// TwinCAT 3 PLC project Ohjaus
// ProgramVersion: 3.1.4024.0
// libraries:
//   Tc2_Standard, * (Beckhoff Automation GmbH)
//   Tc2_System, * (Beckhoff Automation GmbH)
//   Tc3_Module, * (Beckhoff Automation GmbH)
//   VisuSymbols,3.5.10.0,System
// project tree:
//   / GlobalTextList.TcGTLO, PlcTask.TcTTO, Visualization Manager.TcVMO (not stored)
//   GVLs/ GVL.TcGVL, GVL_safety.TcGVL
//   POUs/ MAIN.TcPOU
//   POUs/Modules/ Handling.TcPOU, PickandPlace.TcPOU, Separating.TcPOU, Visu_handling.TcPOU, Sorting.TcPOU
//   VISUs/ Visualization.TcVIS
// real-time tasks:
//   TASK PlcTask: cycle T#10ms, priority 20, ADS port 350
// I/O:
//   DEVICE Device 1 (EtherCAT), AmsNetId 5.59.45.73.2.1
//     Term 1 (EK1200) [EK1200-5000 EtherCAT Power supply (2A E-Bus)]
//       Term 2 (EL1809) [EL1809 16Ch. Dig. Input 24V, 3ms]
//       Term 3 (EL2809) [EL2809 16Ch. Dig. Output 24V, 0.5A]
//       Term 4 (EL4021) [EL4021 1Ch. Ana. Output 4-20mA, 12bit]
//       Term 5 (EL3061) [EL3061 1Ch. Ana. Input 0-10V]
//       Term 6 (EL4021) [EL4021 1Ch. Ana. Output 4-20mA, 12bit]
//       Term 7 (EL2809) [EL2809 16Ch. Dig. Output 24V, 0.5A]
//       Term 8 (EL1809) [EL1809 16Ch. Dig. Input 24V, 3ms]
//       Term 9 (EL6900) [EL6900, TwinSAFE PLC]
//       Term 10 (EL1904) [EL1904, 4 Ch. Safety Input 24V, TwinSAFE]
//         modules: Module 1 (FSOES)
//       Term 11 (EL2904) [EL2904, 4 Ch. Safety Output 24V, 0.5A, TwinSAFE]
//         modules: Module 1 (FSOES), Module 2 (DO)
//       Term 12 (EL9011) [EL9011 End Terminal]
//   DEVICE Device 3 (NOV-DP-RAM)
// variable links:
//   Device 1 (EtherCAT) <-> Device 1 (EtherCAT)/Term 1 (EK1200)/Term 10 (EL1904)
//     Term 1 (EK1200)/Term 9 (EL6900)/ConnectionOutputs/Message_5 RxPDO <-> Module 1 (FSOES)/TxPDO/FSOE
//   Device 1 (EtherCAT) <-> Device 1 (EtherCAT)/Term 1 (EK1200)/Term 11 (EL2904)
//     Term 1 (EK1200)/Term 9 (EL6900)/ConnectionOutputs/Message_6 RxPDO <-> Module 1 (FSOES)/TxPDO/FSOE
//   Device 1 (EtherCAT) <-> Device 1 (EtherCAT)/Term 1 (EK1200)/Term 9 (EL6900)
//     Term 1 (EK1200)/Term 10 (EL1904)/Module 1 (FSOES)/RxPDO/FSOE <-> ConnectionInputs/Message_5 TxPDO
//     Term 1 (EK1200)/Term 11 (EL2904)/Module 1 (FSOES)/RxPDO/FSOE <-> ConnectionInputs/Message_6 TxPDO
//   Ohjaus/Ohjaus Instance <-> Device 1 (EtherCAT)/Term 1 (EK1200)/Term 2 (EL1809)
//     PlcTask Inputs/GVL.X1_I0 <-> Channel 9/Input
//     PlcTask Inputs/GVL.X1_I1 <-> Channel 10/Input
//     PlcTask Inputs/GVL.X1_I2 <-> Channel 13/Input
//     PlcTask Inputs/GVL.X1_I3 <-> Channel 14/Input
//     PlcTask Inputs/GVL.X1_I4 <-> Channel 15/Input
//     PlcTask Inputs/GVL.X1_I5 <-> Channel 16/Input
//     PlcTask Inputs/GVL.X1_I6 <-> Channel 1/Input
//     PlcTask Inputs/GVL.X1_I7 <-> Channel 2/Input
//     PlcTask Inputs/GVL.X2_I0 <-> Channel 3/Input
//     PlcTask Inputs/GVL.X2_I1 <-> Channel 4/Input
//     PlcTask Inputs/GVL.X2_I2 <-> Channel 5/Input
//     PlcTask Inputs/GVL.X2_I4 <-> Channel 6/Input
//     PlcTask Inputs/GVL.X2_I5 <-> Channel 7/Input
//     PlcTask Inputs/GVL_safety.Relay1_EDM <-> Channel 11/Input
//     PlcTask Inputs/GVL_safety.Start_button <-> Channel 12/Input
//   Ohjaus/Ohjaus Instance <-> Device 1 (EtherCAT)/Term 1 (EK1200)/Term 3 (EL2809)
//     PlcTask Outputs/GVL.X1_00 <-> Channel 5/Output
//     PlcTask Outputs/GVL.X1_01 <-> Channel 6/Output
//     PlcTask Outputs/GVL.X1_02 <-> Channel 7/Output
//     PlcTask Outputs/GVL.X1_03 <-> Channel 9/Output
//     PlcTask Outputs/GVL.X1_04 <-> Channel 10/Output
//     PlcTask Outputs/GVL.X1_05 <-> Channel 11/Output
//     PlcTask Outputs/GVL.X1_06 <-> Channel 12/Output
//     PlcTask Outputs/GVL.X1_07 <-> Channel 13/Output
//     PlcTask Outputs/GVL.X2_00 <-> Channel 14/Output
//     PlcTask Outputs/GVL.X2_01 <-> Channel 15/Output
//     PlcTask Outputs/GVL.X2_02 <-> Channel 16/Output
//     PlcTask Outputs/GVL.X4_00 <-> Channel 1/Output
//     PlcTask Outputs/GVL.X4_01 <-> Channel 2/Output
//     PlcTask Outputs/GVL.X4_02 <-> Channel 3/Output
//     PlcTask Outputs/GVL.X4_03 <-> Channel 4/Output
//     PlcTask Outputs/GVL.X4_07 <-> Channel 8/Output
//   Ohjaus/Ohjaus Instance <-> Device 1 (EtherCAT)/Term 1 (EK1200)/Term 7 (EL2809)
//     PlcTask Outputs/GVL.Safety_startpulse <-> Channel 6/Output
//     PlcTask Outputs/GVL.X2_03 <-> Channel 9/Output
//     PlcTask Outputs/GVL.X2_04 <-> Channel 10/Output
//     PlcTask Outputs/GVL.X2_05 <-> Channel 11/Output
//     PlcTask Outputs/GVL.X2_06 <-> Channel 12/Output
//     PlcTask Outputs/GVL.X2_07 <-> Channel 13/Output
//     PlcTask Outputs/GVL.X3_00 <-> Channel 1/Output
//     PlcTask Outputs/GVL.X3_01 <-> Channel 2/Output
//     PlcTask Outputs/GVL.X3_02 <-> Channel 3/Output
//     PlcTask Outputs/GVL.X3_03 <-> Channel 4/Output
//     PlcTask Outputs/GVL.X3_04 <-> Channel 5/Output
//     PlcTask Outputs/GVL.X3_06 <-> Channel 7/Output
//     PlcTask Outputs/GVL.X3_07 <-> Channel 8/Output
//   Ohjaus/Ohjaus Instance <-> Device 1 (EtherCAT)/Term 1 (EK1200)/Term 8 (EL1809)
//     PlcTask Inputs/GVL.X2_I6 <-> Channel 9/Input
//     PlcTask Inputs/GVL.X2_I7 <-> Channel 10/Input
//     PlcTask Inputs/GVL.X3_I0 <-> Channel 1/Input
//     PlcTask Inputs/GVL.X3_I1 <-> Channel 2/Input
//     PlcTask Inputs/GVL.X3_I2 <-> Channel 3/Input
//     PlcTask Inputs/GVL.X3_I4 <-> Channel 4/Input
//     PlcTask Inputs/GVL.X3_I5 <-> Channel 5/Input
//     PlcTask Inputs/GVL.X3_I6 <-> Channel 6/Input
//     PlcTask Inputs/GVL.X4_I0 <-> Channel 11/Input
//     PlcTask Inputs/GVL.X4_I1 <-> Channel 12/Input
//     PlcTask Inputs/GVL.X4_I2 <-> Channel 13/Input
//     PlcTask Inputs/GVL.X4_I3 <-> Channel 14/Input
//     PlcTask Inputs/GVL.X4_I4 <-> Channel 15/Input
//     PlcTask Inputs/GVL.X4_I5 <-> Channel 16/Input
//     PlcTask Inputs/GVL_safety.Safety_Restart <-> Channel 8/Input
//     PlcTask Inputs/MAIN.IbEStopReset <-> Channel 7/Input
//   Ohjaus/Ohjaus Instance <-> Device 1 (EtherCAT)/Term 1 (EK1200)/Term 9 (EL6900)
//     PlcTask Inputs/GVL_safety.Com_Err <-> StandardInputs/Standard Out Var 13
//     PlcTask Inputs/GVL_safety.FB_Err <-> StandardInputs/Standard Out Var 12
//     PlcTask Inputs/GVL_safety.Out_Err <-> StandardInputs/Standard Out Var 14
//     PlcTask Inputs/GVL_safety.Start_pulse <-> StandardInputs/Standard Out Var 9
//     PlcTask Inputs/MAIN.IbEStopError <-> StandardInputs/Standard Out Var 10
//     PlcTask Outputs/GVL_safety.Safety_RUNSTOP <-> StandardOutputs/Standard In Var 11
//     PlcTask Outputs/MAIN.QbEStopReset <-> StandardOutputs/Standard In Var 8
//     PlcTask Outputs/MAIN.QbSafetyErrAck <-> StandardOutputs/Standard In Var 2
//     PlcTask Outputs/MAIN.relay1 <-> StandardOutputs/Standard In Var 7

CONFIGURATION Ohjaus
    RESOURCE PLC ON TwinCAT3
        TASK PlcTask(INTERVAL := T#10ms, PRIORITY := 20);
        PROGRAM MAIN WITH PlcTask : MAIN;
        PROGRAM Visu_handling WITH PlcTask : Visu_handling;
        PROGRAM PickandPlace WITH PlcTask : PickandPlace;
        PROGRAM Sorting WITH PlcTask : Sorting;
        PROGRAM Handling WITH PlcTask : Handling;
        PROGRAM Separating WITH PlcTask : Separating;
    END_RESOURCE
END_CONFIGURATION

// ---- GVLs/GVL.TcGVL
{attribute 'qualified_only'}
VAR_GLOBAL
	X1_I0 AT %I* : BOOL; // Part available
	X1_I1 AT %I* : BOOL; // Mini-slide rectracted
	X1_I2 AT %I* : BOOL; // Mini-slide extended
	X1_I3 AT %I* : BOOL; // Mini-slide up
	X1_I4 AT %I* : BOOL; // Workpiece picked up
	X1_I5 AT %I* : BOOL; // Workpiece at processing position
	X1_I6 AT %I* : BOOL; // No workpiece at conveyor end
	X1_I7 AT %I* : BOOL; // Downstream station free
	X2_I0 AT %I* : BOOL; // Workpeace available
	X2_I1 AT %I* : BOOL; // Metallic workpiece
	X2_I2 AT %I* : BOOL; // Workpiece is not black
	X2_I3 AT %I* : BOOL; // Slide full
	X2_I4 AT %I* : BOOL; // Switch 1 redacted
	X2_I5 AT %I* : BOOL; // Switch 1 extended
	X2_I6 AT %I* : BOOL; // Switch 2 retracted
	X2_I7 AT %I* : BOOL; // Switch 2 extended
	X3_I0 AT %I* : BOOL; // Workpiece available
	X3_I1 AT %I* : BOOL; // Handling at upstream station
	X3_I2 AT %I* : BOOL; // Handling at downstream station
	X3_I3 AT %I* : BOOL; // Handling at sorting position
	X3_I4 AT %I* : BOOL; // Gripper extended
	X3_I5 AT %I* : BOOL; // Gripper retracted
	X3_I6 AT %I* : BOOL; // Workpiece is not black
	X3_I7 AT %I* : BOOL; // 
	X4_I0 AT %I* : BOOL; // Workpiece awailable
	X4_I1 AT %I* : BOOL; // Workpiece at stopper
	X4_I2 AT %I* : BOOL; // Workpiece "housing"
	X4_I3 AT %I* : BOOL; // Switch retracted
	X4_I4 AT %I* : BOOL; // No workpiece on conveyor 2 (buffer empty)
	X4_I5 AT %I* : BOOL; // No Workpiece available at pick-up point
	X4_I6 AT %I* : BOOL; // 
	X4_I7 AT %I* : BOOL; // Downstream station A free
	S1 AT %I* : BOOL; // Kapula S1
	S2 AT %I* : BOOL; // Kapula S2
	S3 AT %I* : BOOL; // Kapula S3
	S4 AT %I* : BOOL; // Kapula S4
	S5 AT %I* : BOOL; // Kapula S5
	S6 AT %I* : BOOL; // Kapula S6
	
	

	X1_00 AT %Q* : BOOL; // Conveyor motor on
	X1_01 AT %Q* : BOOL; // Retract mini-slide
	X1_02 AT %Q* : BOOL; // Extend mini-slide
	X1_03 AT %Q* : BOOL; // move mini-slide downwards
	X1_04 AT %Q* : BOOL; // Vakuum on
	X1_05 AT %Q* : BOOL; // Extend sperator
	X1_06 AT %Q* : BOOL; // NOFunction
	X1_07 AT %Q* : BOOL; // Station occupied
	X2_00 AT %Q* : BOOL; // Conveyor motor on
	X2_01 AT %Q* : BOOL; // Extend switch 1
	X2_02 AT %Q* : BOOL; // Extend switch 2
	X2_03 AT %Q* : BOOL; // Retract stopper
	X2_04 AT %Q* : BOOL; // NOFunction
	X2_05 AT %Q* : BOOL; // NOFunction
	X2_06 AT %Q* : BOOL; // NOFunction
	X2_07 AT %Q* : BOOL; // Station occupied
	X3_00 AT %Q* : BOOL; // Handling to upstream station
	X3_01 AT %Q* : BOOL; // Handling to downstream station
	X3_02 AT %Q* : BOOL; // Extend Gripper
	X3_03 AT %Q* : BOOL; // Open Gripper
	X3_04 AT %Q* : BOOL; //
	X3_05 AT %Q* : BOOL; //
	X3_06 AT %Q* : BOOL; //
	X3_07 AT %Q* : BOOL; // Station occupied
	X4_00 AT %Q* : BOOL; // Conveyor motor 1 on
	X4_01 AT %Q* : BOOL; // Conveyor motor 2 on
	X4_02 AT %Q* : BOOL; // Retract stopper
	X4_03 AT %Q* : BOOL; // Extend switch
	X4_04 AT %Q* : BOOL; //
	X4_05 AT %Q* : BOOL; //
	X4_06 AT %Q* : BOOL; //
	X4_07 AT %Q* : BOOL; // Station occupied
	Safety_startpulse AT %Q* : BOOL;
	VisuIN10 : BOOL;
	VisuIN11 : BOOL;
	VisuIN12 : BOOL;
	VisuIN13 : BOOL;
	VisuIN14 : BOOL;
	VisuIN15 : BOOL;
	VisuIN16 : BOOL;
	VisuIN17 : BOOL;
	VisuIN20 : BOOL;
	VisuIN21 : BOOL;
	VisuIN22 : BOOL;
	VisuIN23 : BOOL;
	VisuIN24 : BOOL;
	VisuIN25 : BOOL;
	VisuIN26 : BOOL;
	VisuIN27 : BOOL;
	VisuIN30 : BOOL;
	VisuIN31 : BOOL;
	VisuIN32 : BOOL;
	VisuIN33 : BOOL;
	VisuIN34 : BOOL;
	VisuIN35 : BOOL;
	VisuIN36 : BOOL;
	VisuIN37 : BOOL;
	VisuOUT0 : BOOL;
	VisuOUT1 : BOOL;
	VisuOUT2 : BOOL;
	VisuOUT3 : BOOL;
	VisuOUT4 : BOOL;
	VisuOUT5 : BOOL;
	VisuOUT6 : BOOL;
	VisuOUT7 : BOOL;
	VisuOUT20 : BOOL;
	VisuOUT21 : BOOL;
	VisuOUT22 : BOOL;
	VisuOUT23 : BOOL;
	VisuOUT24 : BOOL;
	VisuOUT25 : BOOL;
	VisuOUT26 : BOOL;
	VisuOUT27 : BOOL;
	VisuOUT30: BOOL;
	VisuOUT31 : BOOL;
	VisuOUT32: BOOL;
	VisuOUT33 : BOOL;
	VisuOUT34 : BOOL;
	VisuOUT35: BOOL;
	VisuOUT36 : BOOL;
	VisuOUT37 : BOOL;
END_VAR

// ---- GVLs/GVL_safety.TcGVL
{attribute 'qualified_only'}
VAR_GLOBAL
	Safety_RUNSTOP AT %Q* : BOOL;
	FB_Err AT%I* : BOOL;
	Com_Err AT%I* : BOOL;
	Out_Err AT%I* : BOOL;
	Safety_Restart AT%I* :BOOL;
	Relay1_EDM AT%I* :BOOL;
	Start_button AT%I* :BOOL;
	
	Start_pulse AT %I* :BOOL;
	
END_VAR

// ---- POUs/MAIN.TcPOU
PROGRAM MAIN
VAR
	Status_active : BOOL;
		//To safety alias devices
	QbSafetyErrAck  AT%Q* : BOOL := FALSE;
	QbEStopReset    AT%Q* : BOOL;
	bQSafetyRun     AT%Q* : BOOL;
	bQEStopEDM      AT%Q* : BOOL;
	relay1 			AT%Q* : BOOL;
	relay2			AT%Q* : BOOL;
	bQSafetyStartpulse      AT%Q* : BOOL := GVL.Safety_startpulse;
	
	//from safety terminal
	IbEStopReset    AT%I* : BOOL;
	IbEStopEDM      AT%I* : BOOL;
	IbEStopError 	AT%I* : BOOL;
	
	fbDelay 		  	  : TON;
END_VAR

bQEStopEDM := IbEStopEDM;
QbEStopReset := GVL_safety.Safety_Restart;
relay1 := GVL_safety.Relay1_EDM;
bQSafetyRun :=TRUE;
GVL_safety.Safety_RUNSTOP:= TRUE;
IF bQSafetyRun THEN
	QbSafetyErrAck := TRUE;
	fbDelay(IN:=TRUE , PT:=T#75MS , Q=> , ET=> );
	IF fbDelay.Q THEN
		QbSafetyErrAck := FALSE;
	END_IF
END_IF

END_PROGRAM

// ---- POUs/Modules/Visu_handling.TcPOU
PROGRAM Visu_handling
VAR
END_VAR

(*IF GVL.visuOUT0 THEN
	GVL.X1_00 := TRUE;
ELSIF NOT GVL.visuOUT0 THEN
	GVL.X1_00 := FALSE;
END_IF
IF GVL.visuOUT1 THEN
	GVL.X1_01 := TRUE;
ELSIF NOT GVL.visuOUT1 THEN
	GVL.X1_01 := FALSE;
END_IF
IF GVL.visuOUT2 THEN
	GVL.X1_02 := TRUE;
ELSIF NOT GVL.visuOUT2 THEN
	GVL.X1_02 := FALSE;
END_IF
IF GVL.visuOUT3 THEN
	GVL.X1_03 := TRUE;
ELSIF NOT GVL.visuOUT3 THEN
	GVL.X1_03 := FALSE;
END_IF
IF GVL.visuOUT4 THEN
	GVL.X1_04 := TRUE;
ELSIF NOT GVL.visuOUT4 THEN
	GVL.X1_04 := FALSE;
END_IF
IF GVL.visuOUT5 THEN
	GVL.X1_05 := TRUE;
ELSIF NOT GVL.visuOUT5 THEN
	GVL.X1_05 := FALSE;
END_IF
IF GVL.visuOUT6 THEN
	GVL.X1_06 := TRUE;
ELSIF NOT GVL.visuOUT6 THEN
	GVL.X1_06 := FALSE;
END_IF
IF GVL.visuOUT7 THEN
	GVL.X1_07 := TRUE;
ELSIF NOT GVL.visuOUT7 THEN
	GVL.X1_07 := FALSE;
END_IF


IF GVL.visuOUT20 THEN
	GVL.X2_00 := TRUE;
ELSIF NOT GVL.visuOUT20 THEN
	GVL.X2_00 := FALSE;
END_IF
IF GVL.visuOUT21 THEN
	GVL.X2_01 := TRUE;
ELSIF NOT GVL.visuOUT21 THEN
	GVL.X2_01 := FALSE;
END_IF
IF GVL.visuOUT22 THEN
	GVL.X2_02 := TRUE;
ELSIF NOT GVL.visuOUT22 THEN
	GVL.X2_02 := FALSE;
END_IF
IF GVL.visuOUT23 THEN
	GVL.X2_03 := TRUE;
ELSIF NOT GVL.visuOUT23 THEN
	GVL.X2_03 := FALSE;
END_IF*)

END_PROGRAM

// ---- POUs/Modules/PickandPlace.TcPOU
PROGRAM PickandPlace
VAR
	Station_occupied : BOOL;
	Timerdelay0 : TON;
	Start_timer0 : BOOL;
	Statustimer0 : BOOL;
	Timerdelay1 : TON;
	Start_timer1 : BOOL;
	Statustimer1 : BOOL;
	Start_timer2 : BOOL;
	Timerdelay2 : TON;
	Statustimer2 : BOOL;
	Start_timer3 : BOOL;
	Timerdelay3 : TP;
	Statustimer3 : BOOL;
	Start_timer4 : BOOL;
	Timerdelay4 : TON;
	Statustimer4 : BOOL;
	PICKUP_STEP : INT;
END_VAR

Timerdelay0(IN := Start_timer0 , PT:=  T#1000MS , Q =>Statustimer0);
Timerdelay1(IN := Start_timer1 , PT:=  T#1000MS , Q =>Statustimer1);
Timerdelay2(IN := Start_timer2 , PT:=  T#1000MS , Q =>Statustimer2);
Timerdelay3(IN := Start_timer3 , PT:=  T#800MS , Q =>Statustimer3);
Timerdelay4(IN := Start_timer4 , PT:=  T#800MS , Q =>Statustimer4);

		IF GVL.X1_I0 AND Station_occupied = FALSE THEN //Check if piece is available
		GVL.X1_00 := TRUE; //Turn on conveyor belt
		GVL.X2_00 := TRUE;
		GVL.X4_00 := TRUE;
		Start_timer0 := FALSE;		
		Start_timer1 := FALSE;
		Start_timer2 := FALSE;
		Statustimer0 := FALSE;
		Statustimer1 := FALSE;
		Statustimer2 := FALSE;
		Start_timer3 := FALSE;
		Start_timer4 := FALSE;
		Statustimer3 := FALSE;
		Statustimer4 := FALSE;
		PICKUP_STEP:=1;
		END_IF
		CASE PICKUP_STEP OF
			1:
		Station_occupied := TRUE;
		Start_timer0 := TRUE;
		GVL.X1_01 := TRUE;  //Retract mini-slide
		
		IF GVL.X1_I1 = TRUE AND Statustimer0 = TRUE THEN //Check if retracted
			Start_timer0 := FALSE;
			PICKUP_STEP:=2;
		END_IF
			2:
		GVL.X1_03 := TRUE;  //move mini-slide downwards
		Start_timer1 :=TRUE;

		IF Statustimer1 THEN
			Start_timer1 := FALSE;
			PICKUP_STEP:=3;
		END_IF
			3:
		GVL.X1_04 := TRUE; // Vacuum on 
		PICKUP_STEP:=4;
			4:
		GVL.X1_03 := FALSE; //move mini-slide upwards
		Start_timer2 := TRUE;

		IF Statustimer2 THEN
			Start_timer2 := FALSE;
			PICKUP_STEP:=5;
			END_IF
			5:
		GVL.X1_01 := FALSE; // Turn off retraction of mini-slide
		GVL.X1_02 := TRUE; // Extend mini-slide
		Start_timer2 := FALSE;
		Statustimer2 := FALSE;
		IF GVL.X1_I2 THEN
			PICKUP_STEP:=6;
		END_IF
			6:
		GVL.X1_03 := TRUE; //Move mini-slide downwards
		Start_timer3 := TRUE;

		IF Statustimer3 THEN
		Start_timer3 := FALSE;
		GVL.X1_04 := FALSE; // Vacuum off
		GVL.X1_03 := FALSE;  //Move mini-slide upwards
		Start_timer4 := TRUE;
		END_IF
		IF Statustimer4 THEN
		Start_timer4 := TRUE;
		Station_occupied := FALSE;
		GVL.X1_02 := FALSE;
		PICKUP_STEP := 0;
		END_IF
		0:
			//Wait until new cycle.
			 
		END_CASE

END_PROGRAM

// ---- POUs/Modules/Sorting.TcPOU
PROGRAM Sorting
VAR
	
	Timerdelay0 : TON;
	Statustimer0 : BOOL;
	Timerdelay1 : TON;
	Statustimer1 : BOOL;
	Timerdelay2 : TON;
	Statustimer2 : BOOL;
	Timerdelay3 : TON;
	Statustimer3 : BOOL;
END_VAR

Timerdelay0(PT:=  T#5000MS , Q =>Statustimer0);
Timerdelay1(PT:=  T#1000MS , Q =>Statustimer1);
Timerdelay2(PT:=  T#1000MS , Q =>Statustimer2);
Timerdelay3(PT:=  T#800MS , Q =>Statustimer3);

(*
Do not turn conveyor on when GVL.X2_I3 slide is full 

IF GVL.X2_I0 THEN
	GVL.X2_00 := TRUE;
	END_IF
	IF Statustimer0 THEN
		GVL.X2_00 := FALSE;
	END_IF
	


Metallic workpiece (X2_I1) Wait and turn conveyor on then
 turn slide 1. 



*)

END_PROGRAM

// ---- POUs/Modules/Handling.TcPOU
PROGRAM Handling
VAR
	Station_occupied : BOOL;
	Timerdelay0 : TON;
	Statustimer0 : BOOL;
	Timerdelay1 : TON;
	Statustimer1 : BOOL;
	Timerdelay2 : TON;
	Statustimer2 : BOOL;
	Timerdelay3 : TON;
	Statustimer3 : BOOL;
	Timerdelay4 : TON;
	Statustimer4 : BOOL;
	PICKUP_STEP : INT;
END_VAR

Timerdelay0( PT:=  T#1800MS , Q =>Statustimer0);
Timerdelay1( PT:=  T#1200MS , Q =>Statustimer1);
Timerdelay2( PT:=  T#1800MS , Q =>Statustimer2);
Timerdelay3( PT:=  T#1400MS , Q =>Statustimer3);
Timerdelay4(PT:=  T#900MS , Q =>Statustimer4);
		IF GVL.X3_I0 AND Station_occupied = FALSE THEN //Check if piece is awailable

		Statustimer0 := FALSE;
		Statustimer1 := FALSE;
		Statustimer2 := FALSE;
		Statustimer3 := FALSE;
		Statustimer4 := FALSE;
		PICKUP_STEP:=1;
		END_IF

		CASE PICKUP_STEP OF
			1:
		Station_occupied := TRUE;
		Timerdelay0.IN:=TRUE;
		GVL.X3_00 := TRUE;  //Handling to downstream station
		
		IF  Statustimer0 = TRUE THEN
			Timerdelay0.IN:= FALSE;
			PICKUP_STEP:=2;
		END_IF
			2:
		GVL.X3_02 := TRUE;  //Extend gripper
		Timerdelay1.IN:=TRUE;

		IF Statustimer1 THEN
			Timerdelay1.IN:=FALSE;
			PICKUP_STEP:=3;
		END_IF
			3:
		GVL.X3_03 := TRUE; // Close Gripper
		PICKUP_STEP:=4;
			4:
		GVL.X3_02 := FALSE; // Move gripper upwards
		Timerdelay2.IN:=TRUE;

		IF Statustimer2 THEN
			Timerdelay2.IN:=FALSE;
			PICKUP_STEP:=5;
			END_IF
			5:
		GVL.X3_00 := FALSE; // 
		GVL.X3_01 := TRUE; // 
		IF GVL.X3_I4 THEN
			PICKUP_STEP:=6;
		END_IF
			6:
		GVL.X3_02 := TRUE; //Extend gripper
		Timerdelay3.IN:=TRUE;

		IF Statustimer3 THEN
		Timerdelay3.IN:=FALSE;
		GVL.X3_02 := FALSE;
		Timerdelay4.IN:=TRUE;
		END_IF
		IF Statustimer4 THEN
		Timerdelay4.IN:=FALSE;
		GVL.X3_02 := FALSE;
		GVL.X3_03 := FALSE; // Open gripper
		GVL.X3_01 :=FALSE;
		GVL.X3_00 := FALSE;
		PICKUP_STEP := 0;
		Station_occupied := FALSE;
		END_IF
		0:
			IF GVL.X3_I0 AND Station_occupied = FALSE THEN
				;
			END_IF
			//Wait until new cycle.
			 
		END_CASE

END_PROGRAM

// ---- POUs/Modules/Separating.TcPOU
PROGRAM Separating
VAR
	Station_occupied : BOOL;	
	Timerdelay0 : TON;
	Start_timer0 : BOOL;
	Statustimer0 : BOOL;
	Timerdelay1 : TON;
	Start_timer1 : BOOL;
	Statustimer1 : BOOL;
	Start_timer2 : BOOL;
	Timerdelay2 : TP;
	Statustimer2 : BOOL;
	Timerdelay3 : TP;
	Start_timer3 : BOOL;
	Statustimer3 : BOOL;
END_VAR

Timerdelay0(IN := Start_timer0 , PT:=  T#1000MS , Q =>Statustimer0);
Timerdelay1(IN := Start_timer1 , PT:=  T#1000MS , Q =>Statustimer1);
Timerdelay2(IN := Start_timer2 , PT:=  T#1000MS , Q =>Statustimer2);
Timerdelay3(IN := Start_timer3 , PT:=  T#800MS , Q =>Statustimer3);
		IF GVL.X1_I0 AND Station_occupied = FALSE THEN //Check if piece is available
				GVL.X1_00 := TRUE; //Turn on conveyor belt
		END_IF

END_PROGRAM

// ---- GlobalTextList.TcGTLO
TEXTLIST GlobalTextList
  9 = 'Conveyor motor on'
  860 = 'Downstream station free'
  615 = 'Extend mini-slide'
  317 = 'Extend mini-slide down'
  24 = 'Extend seperator'
  369 = 'Extend switch 1'
  434 = 'Extend switch 2'
  740 = 'l'
  987 = 'Label'
  888 = 'LabelLabel'
  543 = 'metallic workpiece'
  994 = 'Mini-slide extended'
  951 = 'Mini-slide rectracted'
  537 = 'mini-slide up'
  778 = 'move mini-slide down'
  241 = 'No workpiece at conveyor end'
  423 = 'Part awailable'
  764 = 'Retract mini-slide'
  457 = 'Retract stopper'
  429 = 'slide full'
  32 = 'Station occupied'
  11 = 'Switch 1 extended'
  553 = 'Switch 1 redacted'
  183 = 'Switch 2 extended'
  73 = 'Switch 2 retracted'
  120 = 'Vakuum on'
  887 = 'Workpiece at processing position'
  184 = 'Workpiece awailable'
  810 = 'Workpiece is not black'
  560 = 'Workpiece picked up'
  967 = 'X1 Pick&Place'
  937 = 'X2 Pick&Place'
  872 = 'X2 Sorting'
  542 = 'X3 Handling'
END_TEXTLIST

// ---- VISUs/Visualization.TcVIS
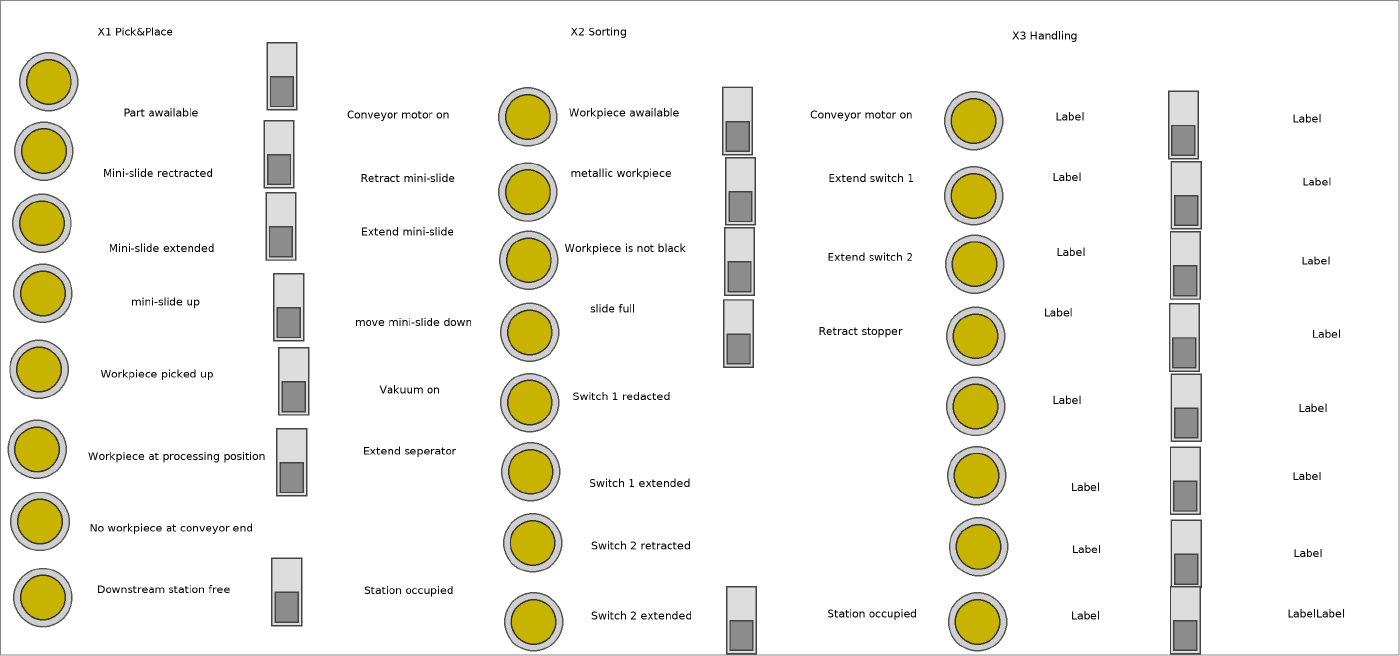
VISUALIZATION Visualization  // 1435x673
    Lamp1 (10,120 70x70), variable: GVL.X1_I1, style: Lamp-Lamp1-Yellow
    DipSwitch (251,123 70x70), variable: GVL.VisuOUT1, behaviour: TOGGLE, style: Switch-DipSwitch-Gray
    Label (64,18 150x30), "X1 Pick&Place"
    Lamp1 (15,49 70x70), variable: GVL.X1_I0, style: Lamp-Lamp1-Yellow
    Lamp1 (8,194 70x70), variable: GVL.X1_I2, style: Lamp-Lamp1-Yellow
    Lamp1 (5,344 70x70), variable: GVL.X1_I4, style: Lamp-Lamp1-Yellow
    Lamp1 (3,426 70x70), variable: GVL.X1_I5, style: Lamp-Lamp1-Yellow
    Lamp1 (6,500 70x70), variable: GVL.X1_I6, style: Lamp-Lamp1-Yellow
    Lamp1 (9,578 70x70), variable: GVL.X1_I7, style: Lamp-Lamp1-Yellow
    DipSwitch (254,43 70x70), variable: GVL.VisuOUT0, behaviour: TOGGLE, style: Switch-DipSwitch-Gray
    DipSwitch (259,572 70x70), variable: GVL.VisuOUT7, behaviour: TOGGLE, style: Switch-DipSwitch-Gray
    DipSwitch (261,280 70x70), variable: GVL.VisuOUT3, behaviour: TOGGLE, style: Switch-DipSwitch-Gray
    DipSwitch (266,356 70x70), variable: GVL.VisuOUT4, behaviour: TOGGLE, style: Switch-DipSwitch-Gray
    DipSwitch (264,439 70x70), variable: GVL.VisuOUT5, behaviour: TOGGLE, style: Switch-DipSwitch-Gray
    Label (90,101 150x30), "Part awailable"
    Label (85,528 182x28), "No workpiece at conveyor end"
    Label (93,590 150x30), "Downstream station free"
    Label (344,591 150x30), "Station occupied"
    Label (345,448 150x30), "Extend seperator"
    Label (345,385 150x30), "Vakuum on"
    Label (349,316 150x30), "move mini-slide down"
    Label (343,168 150x30), "Retract mini-slide"
    Label (333,103 150x30), "Conveyor motor on"
    Label (87,444 188x49), "Workpiece at processing position"
    Label (86,369 150x30), "Workpiece picked up"
    Label (91,240 150x30), "Mini-slide extended"
    Label (87,163 150x30), "Mini-slide rectracted"
    Lamp1 (506,162 70x70), variable: GVL.X2_I1, style: Lamp-Lamp1-Yellow
    DipSwitch (724,161 70x70), variable: GVL.VisuOUT21, behaviour: TOGGLE, style: Switch-DipSwitch-Gray
    Label (539,18 150x30), "X2 Sorting"
    Lamp1 (506,85 70x70), variable: GVL.X2_I0, style: Lamp-Lamp1-Yellow
    Lamp1 (507,232 70x70), variable: GVL.X2_I2, style: Lamp-Lamp1-Yellow
    Lamp1 (508,306 70x70), variable: GVL.X2_I3, style: Lamp-Lamp1-Yellow
    Lamp1 (508,378 70x70), variable: GVL.X2_I4, style: Lamp-Lamp1-Yellow
    Lamp1 (509,449 70x70), variable: GVL.X2_I5, style: Lamp-Lamp1-Yellow
    Lamp1 (511,522 70x70), variable: GVL.X2_I6, style: Lamp-Lamp1-Yellow
    DipSwitch (721,89 70x70), variable: GVL.VisuOUT20, behaviour: TOGGLE, style: Switch-DipSwitch-Gray
    DipSwitch (723,233 70x70), variable: GVL.VisuOUT22, behaviour: TOGGLE, style: Switch-DipSwitch-Gray
    DipSwitch (722,307 70x70), variable: GVL.VisuOUT23, behaviour: TOGGLE, style: Switch-DipSwitch-Gray
    Label (565,101 150x30), "Workpiece awailable"
    Label (581,481 150x30), "Switch 1 extended"
    Label (582,545 150x30), "Switch 2 retracted"
    Label (814,400 150x30)
    Label (807,325 150x30), "Retract stopper"
    Label (817,249 150x30), "Extend switch 2"
    Label (818,168 150x30), "Extend switch 1"
    Label (808,103 150x30), "Conveyor motor on"
    Label (562,392 150x30), "Switch 1 redacted"
    Label (553,302 150x30), "slide full"
    Label (566,240 150x30), "Workpiece is not black"
    Label (562,163 150x30), "metallic workpiece"
    Lamp1 (963,166 70x70), style: Lamp-Lamp1-Yellow
    DipSwitch (1181,165 70x70), behaviour: TOGGLE, style: Switch-DipSwitch-Gray
    Label (996,22 150x30), "X3 Handling"
    Lamp1 (963,89 70x70), style: Lamp-Lamp1-Yellow
    Lamp1 (964,236 70x70), style: Lamp-Lamp1-Yellow
    Lamp1 (965,310 70x70), style: Lamp-Lamp1-Yellow
    Lamp1 (965,382 70x70), style: Lamp-Lamp1-Yellow
    Lamp1 (966,453 70x70), style: Lamp-Lamp1-Yellow
    Lamp1 (968,526 70x70), style: Lamp-Lamp1-Yellow
    DipSwitch (1178,93 70x70), behaviour: TOGGLE, style: Switch-DipSwitch-Gray
    DipSwitch (1181,533 70x70), behaviour: TOGGLE, style: Switch-DipSwitch-Gray
    DipSwitch (1180,237 70x70), behaviour: TOGGLE, style: Switch-DipSwitch-Gray
    DipSwitch (1179,311 70x70), behaviour: TOGGLE, style: Switch-DipSwitch-Gray
    DipSwitch (1181,383 70x70), behaviour: TOGGLE, style: Switch-DipSwitch-Gray
    DipSwitch (1180,458 70x70), behaviour: TOGGLE, style: Switch-DipSwitch-Gray
    Label (1022,105 150x30), "Label"
    Label (1038,485 150x30), "Label"
    Label (1039,549 150x30), "Label"
    Label (1266,553 150x30), "Label"
    Label (1265,474 150x30), "Label"
    Label (1271,404 150x30), "Label"
    Label (1285,328 150x30), "Label"
    Label (1274,253 150x30), "Label"
    Label (1275,172 150x30), "Label"
    Label (1265,107 150x30), "Label"
    Label (1019,396 150x30), "Label"
    Label (1010,306 150x30), "Label"
    Label (1023,244 150x30), "Label"
    Label (1019,167 150x30), "Label"
    Lamp1 (9,266 70x70), variable: GVL.X1_I3, style: Lamp-Lamp1-Yellow
    Label (95,295 150x30), "mini-slide up"
    DipSwitch (253,197 70x70), variable: GVL.VisuOUT2, behaviour: TOGGLE, style: Switch-DipSwitch-Gray
    Label (343,223 150x30), "Extend mini-slide"
    DipSwitch (725,601 70x70), variable: GVL.VisuOUT27, behaviour: TOGGLE, style: Switch-DipSwitch-Gray
    Label (583,617 150x30), "Switch 2 extended"
    Lamp1 (512,603 70x70), variable: GVL.X2_I7, style: Lamp-Lamp1-Yellow
    Label (819,615 150x30), "Station occupied"
    DipSwitch (1180,601 70x70), behaviour: TOGGLE, style: Switch-DipSwitch-Gray
    Label (1038,617 150x30), "Label"
    Lamp1 (967,603 70x70), style: Lamp-Lamp1-Yellow
    Label (1274,615 150x30), "LabelLabel"
END_VISUALIZATION
